PROGRAM MAIN
VAR
	stDemo	: ST_Demo;
	stArrayDemo	: ARRAY[1..100]OF ST_Demo;
	
	i: INT;
	
END_VAR

IF bInput1	THEN
	FOR i:= 0 TO 100 DO
		stArrayDemo[i+1].nVar	:= i*i;
		stArrayDemo[i+1].fVar	:= INT_TO_LREAL(i)+1.345;
	END_FOR
END_IF

ACT_Motion();

PRG_Servo1();

ACTION ACT_Motion:
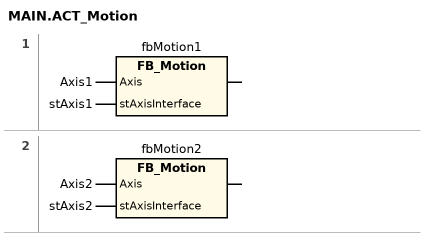
// NETWORK 1
fbMotion1(Axis := Axis1, stAxisInterface := stAxis1); // FB_Motion

// NETWORK 2
fbMotion2(Axis := Axis2, stAxisInterface := stAxis2); // FB_Motion
END_ACTION

END_PROGRAM

(* stored: Version 1.1.0.1, ProductVersion 3.1.4022.12
   POU MAIN: Id {7f3c4b9b-e12a-4a4f-a3c2-3466a897f79b}, SpecialFunc None
   Action ACT_Motion: Id {ea6de3bc-710a-496e-930d-be44d4e33e94} *)
